Staubli VAL3: getNum.pgx

public program getNum(num nX, num nY, string sFormat, num& nValue)
  local num i
  local num n
  local string s
begin
  // Acquires a number
  //
  // copyright (c) 2013-2021 victortorreslopez
  //
  // GNU General Public License
  //
  // Parameters
  // - nX: cursor column (0 to 39)
  // - nY: cursor row (0 to 13)
  // - sFormat: display format
  // - &nValue: numerical variable to be set
  //
  // Local variables
  // - i: iterator index
  // - n: number of characters in nValue
  // - s: a string
  //
  // Version history
  // ---------------
  // 0.1, 2021/12/30, VTL: 1s update (coding style)
  // 0.0, 2013/12/10, VTL: alfa release

  // Fills s with spaces
  s = ""
  n = len(toString(sFormat, nValue))
  for i = 0 to n - 1
    s = s + " "
  endFor

  // Displays spaces before acquires the new string value
  gotoxy(nX, nY)
  put(s)

  // Acquires the new numerical value
  gotoxy(nX, nY)
  get(nValue)
end
